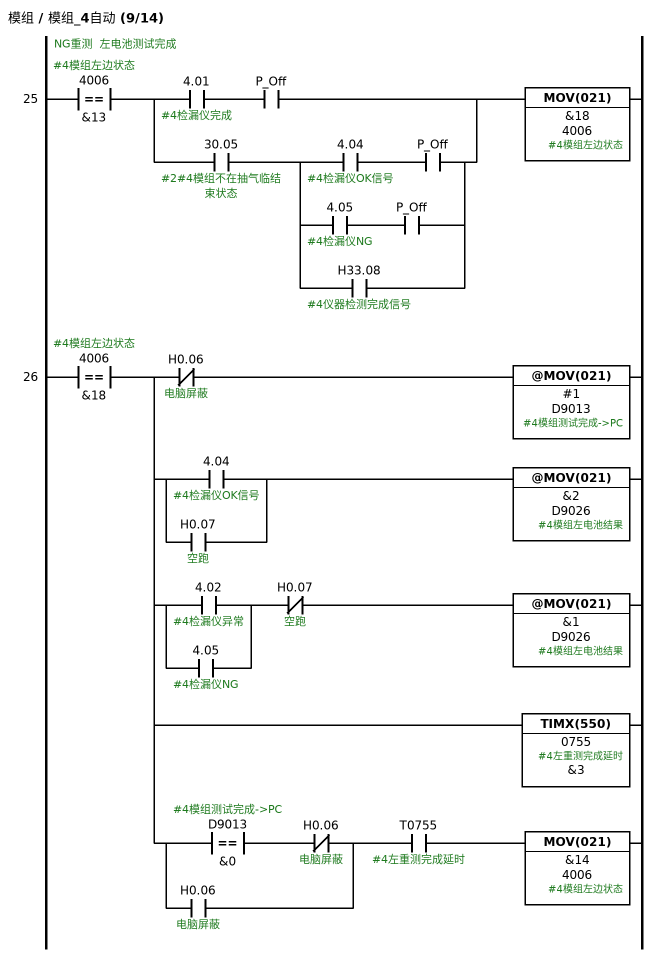
; [picture p257: 模组 / 模组_4自动, rungs 25-26]
; rung 25: NG重测  左电池测试完成
LD=(300) 4006 &13  ; #4模组左边状态
LD 4.01  ; #4检漏仪完成
AND P_Off
LD 30.05  ; #2#4模组不在抽气临结束状态  // 2018/5/29hy修改,所有模组不在临抽气结束状态下，测试模组测试完成后，给出停止测试信号
LD 4.04  ; #4检漏仪OK信号
AND P_Off
LD 4.05  ; #4检漏仪NG
AND P_Off
ORLD
OR H33.08  ; #4仪器检测完成信号
ANDLD
ORLD
ANDLD
MOV(021) &18 4006  ; #4模组左边状态
; rung 26
LD=(300) 4006 &18  ; #4模组左边状态
OUT TR0
ANDNOT H0.06  ; 电脑屏蔽
@MOV(021) #1 D9013  ; #4模组测试完成->PC
LD TR0
LD 4.04  ; #4检漏仪OK信号
OR H0.07  ; 空跑
ANDLD
@MOV(021) &2 D9026  ; #4模组左电池结果
LD TR0
LD 4.02  ; #4检漏仪异常
OR 4.05  ; #4检漏仪NG
ANDLD
ANDNOT H0.07  ; 空跑
@MOV(021) &1 D9026  ; #4模组左电池结果
LD TR0
TIMX(550) 0755 &3  ; #4左重测完成延时
LD=(300) D9013 &0  ; #4模组测试完成->PC
ANDNOT H0.06  ; 电脑屏蔽
OR H0.06  ; 电脑屏蔽
ANDLD
AND T0755  ; #4左重测完成延时
MOV(021) &14 4006  ; #4模组左边状态

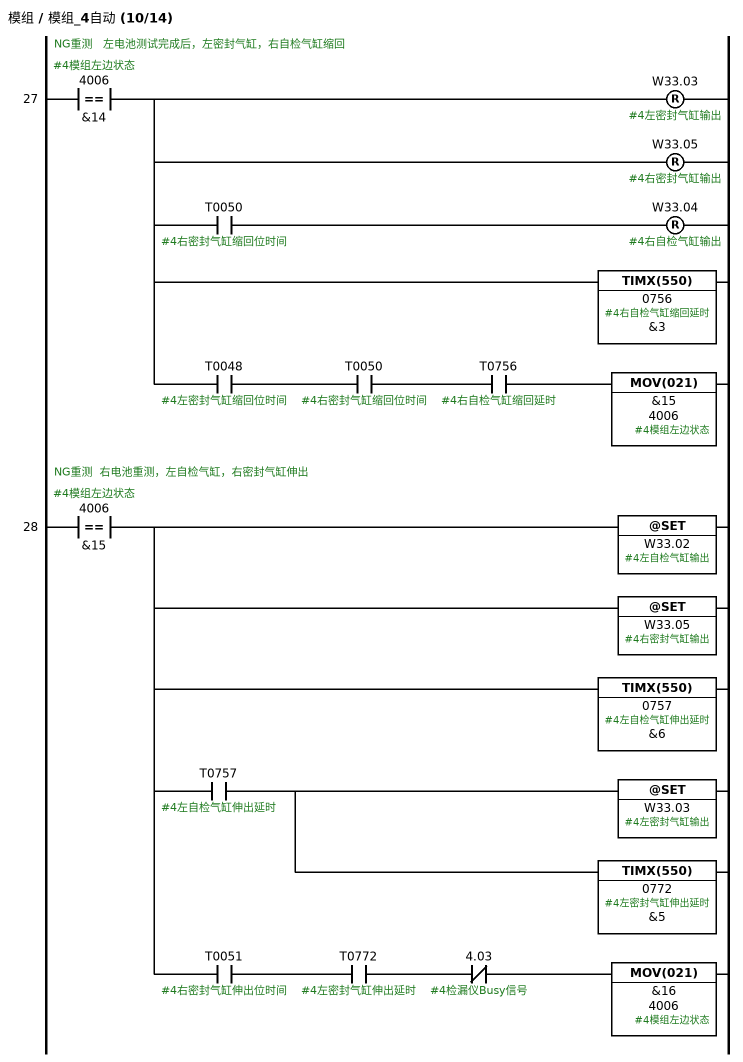
; rung 27: NG重测   左电池测试完成后，左密封气缸，右自检气缸缩回
LD=(300) 4006 &14  ; #4模组左边状态
OUT TR0
RSET W33.03  ; #4左密封气缸输出
RSET W33.05  ; #4右密封气缸输出
AND T0050  ; #4右密封气缸缩回位时间
RSET W33.04  ; #4右自检气缸输出
LD TR0
TIMX(550) 0756 &3  ; #4右自检气缸缩回延时
AND T0048  ; #4左密封气缸缩回位时间
AND T0050  ; #4右密封气缸缩回位时间
AND T0756  ; #4右自检气缸缩回延时
MOV(021) &15 4006  ; #4模组左边状态
; rung 28: NG重测  右电池重测，左自检气缸，右密封气缸伸出
LD=(300) 4006 &15  ; #4模组左边状态
OUT TR0
@SET W33.02  ; #4左自检气缸输出
@SET W33.05  ; #4右密封气缸输出
TIMX(550) 0757 &6  ; #4左自检气缸伸出延时
AND T0757  ; #4左自检气缸伸出延时
@SET W33.03  ; #4左密封气缸输出
TIMX(550) 0772 &5  ; #4左密封气缸伸出延时
LD TR0
AND T0051  ; #4右密封气缸伸出位时间
AND T0772  ; #4左密封气缸伸出延时
ANDNOT 4.03  ; #4检漏仪Busy信号
MOV(021) &16 4006  ; #4模组左边状态

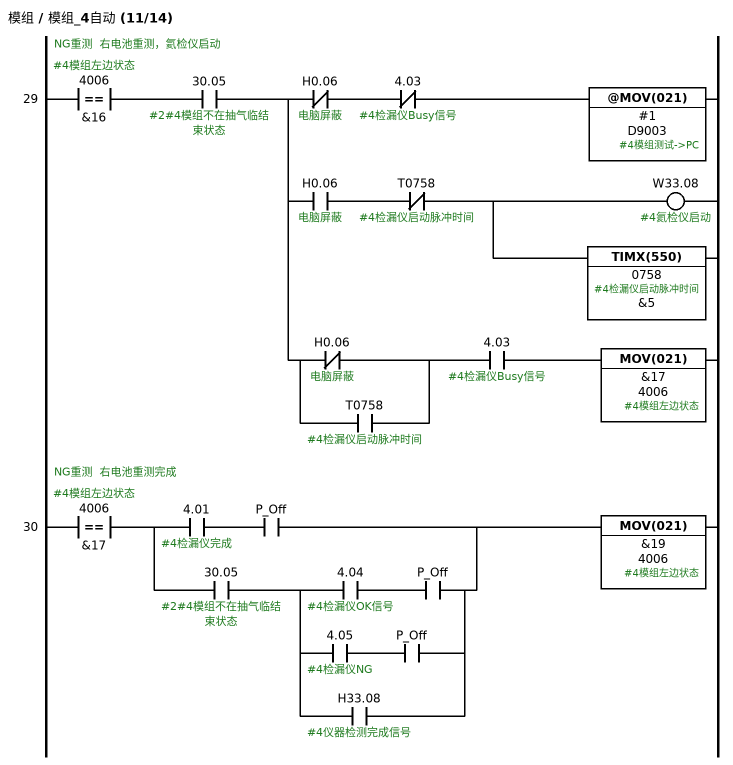
; rung 29: NG重测  右电池重测，氦检仪启动
LD=(300) 4006 &16  ; #4模组左边状态
AND 30.05  ; #2#4模组不在抽气临结束状态  // 2018/5/28hy修改 所有模组不在抽气临结束状态下，下一模组才能启动(防抽气NG)
OUT TR0
ANDNOT H0.06  ; 电脑屏蔽
ANDNOT 4.03  ; #4检漏仪Busy信号
@MOV(021) #1 D9003  ; #4模组测试->PC
LD TR0
AND H0.06  ; 电脑屏蔽
ANDNOT T0758  ; #4检漏仪启动脉冲时间
OUT W33.08  ; #4氦检仪启动
TIMX(550) 0758 &5  ; #4检漏仪启动脉冲时间
LD TR0
LDNOT H0.06  ; 电脑屏蔽
OR T0758  ; #4检漏仪启动脉冲时间
ANDLD
AND 4.03  ; #4检漏仪Busy信号
MOV(021) &17 4006  ; #4模组左边状态
; rung 30: NG重测  右电池重测完成
LD=(300) 4006 &17  ; #4模组左边状态
LD 4.01  ; #4检漏仪完成
AND P_Off
LD 30.05  ; #2#4模组不在抽气临结束状态
LD 4.04  ; #4检漏仪OK信号
AND P_Off
LD 4.05  ; #4检漏仪NG
AND P_Off
ORLD
OR H33.08  ; #4仪器检测完成信号
ANDLD
ORLD
ANDLD
MOV(021) &19 4006  ; #4模组左边状态

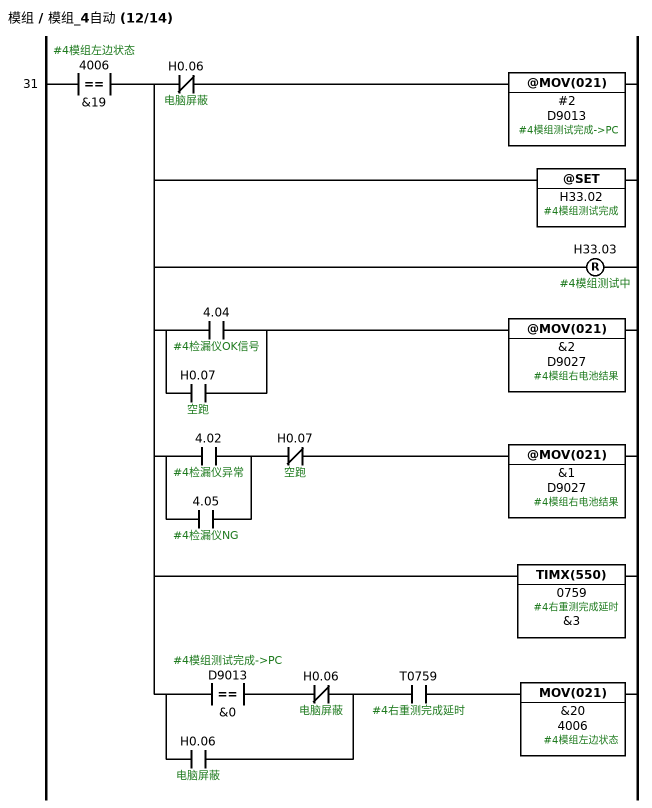
; rung 31
LD=(300) 4006 &19  ; #4模组左边状态
OUT TR0
ANDNOT H0.06  ; 电脑屏蔽
@MOV(021) #2 D9013  ; #4模组测试完成->PC
LD TR0
@SET H33.02  ; #4模组测试完成
RSET H33.03  ; #4模组测试中
LD 4.04  ; #4检漏仪OK信号
OR H0.07  ; 空跑
ANDLD
@MOV(021) &2 D9027  ; #4模组右电池结果
LD TR0
LD 4.02  ; #4检漏仪异常
OR 4.05  ; #4检漏仪NG
ANDLD
ANDNOT H0.07  ; 空跑
@MOV(021) &1 D9027  ; #4模组右电池结果
LD TR0
TIMX(550) 0759 &3  ; #4右重测完成延时
LD=(300) D9013 &0  ; #4模组测试完成->PC
ANDNOT H0.06  ; 电脑屏蔽
OR H0.06  ; 电脑屏蔽
ANDLD
AND T0759  ; #4右重测完成延时
MOV(021) &20 4006  ; #4模组左边状态

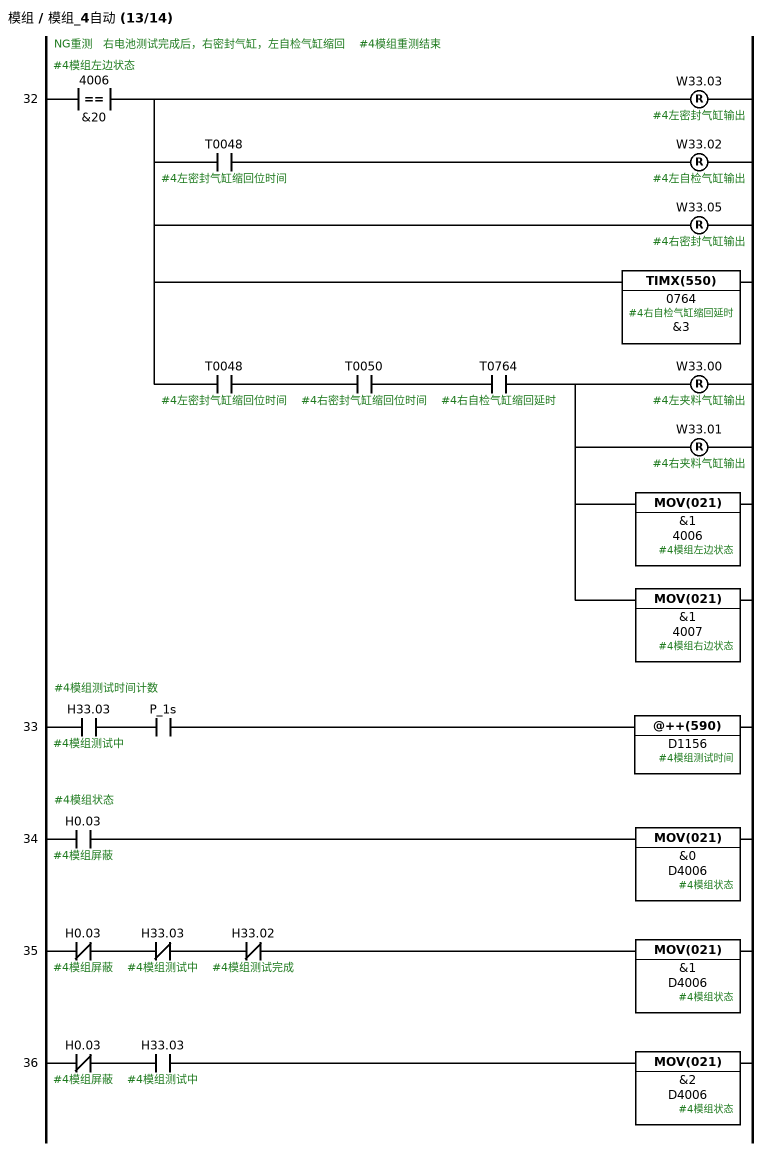
; rung 32: NG重测   右电池测试完成后，右密封气缸，左自检气缸缩回    #4模组重测结束
LD=(300) 4006 &20  ; #4模组左边状态
OUT TR0
RSET W33.03  ; #4左密封气缸输出
AND T0048  ; #4左密封气缸缩回位时间
RSET W33.02  ; #4左自检气缸输出
LD TR0
RSET W33.05  ; #4右密封气缸输出
TIMX(550) 0764 &3  ; #4右自检气缸缩回延时
AND T0048  ; #4左密封气缸缩回位时间
AND T0050  ; #4右密封气缸缩回位时间
AND T0764  ; #4右自检气缸缩回延时
RSET W33.00  ; #4左夹料气缸输出
RSET W33.01  ; #4右夹料气缸输出
MOV(021) &1 4006  ; #4模组左边状态
MOV(021) &1 4007  ; #4模组右边状态
; rung 33: #4模组测试时间计数
LD H33.03  ; #4模组测试中
AND P_1s
@++(590) D1156  ; #4模组测试时间
; rung 34: #4模组状态
LD H0.03  ; #4模组屏蔽
MOV(021) &0 D4006  ; #4模组状态
; rung 35
LDNOT H0.03  ; #4模组屏蔽
ANDNOT H33.03  ; #4模组测试中
ANDNOT H33.02  ; #4模组测试完成
MOV(021) &1 D4006  ; #4模组状态
; rung 36
LDNOT H0.03  ; #4模组屏蔽
AND H33.03  ; #4模组测试中
MOV(021) &2 D4006  ; #4模组状态

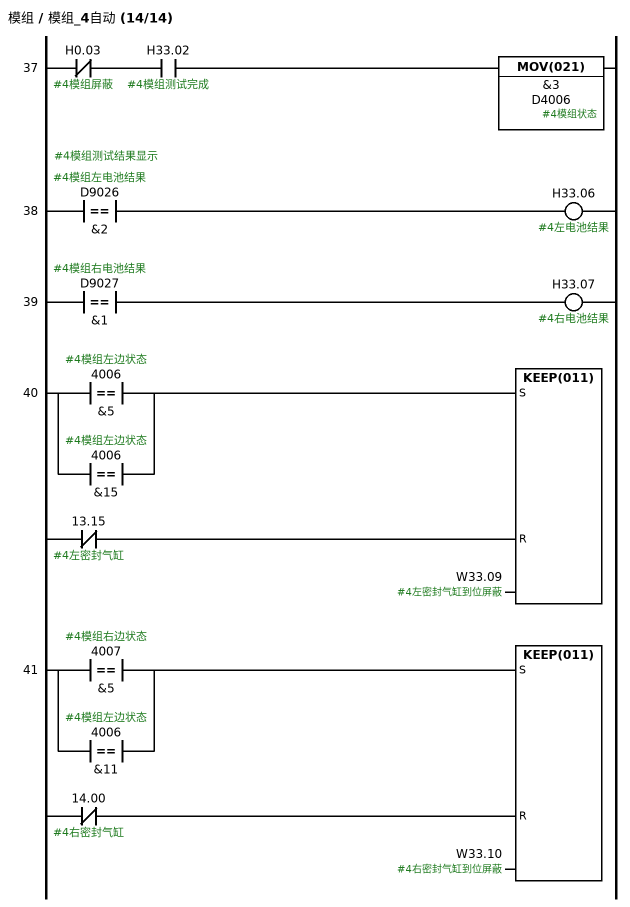
; rung 37
LDNOT H0.03  ; #4模组屏蔽
AND H33.02  ; #4模组测试完成
MOV(021) &3 D4006  ; #4模组状态
; rung 38: #4模组测试结果显示
LD=(300) D9026 &2  ; #4模组左电池结果
OUT H33.06  ; #4左电池结果
; rung 39
LD=(300) D9027 &1  ; #4模组右电池结果
OUT H33.07  ; #4右电池结果
; rung 40
LD=(300) 4006 &5  ; #4模组左边状态
OR=(300) 4006 &15  ; #4模组左边状态
LDNOT 13.15  ; #4左密封气缸
KEEP(011) W33.09  ; #4左密封气缸到位屏蔽
; rung 41
LD=(300) 4007 &5  ; #4模组右边状态
OR=(300) 4006 &11  ; #4模组左边状态
LDNOT 14.00  ; #4右密封气缸
KEEP(011) W33.10  ; #4右密封气缸到位屏蔽

### Section 外部输出

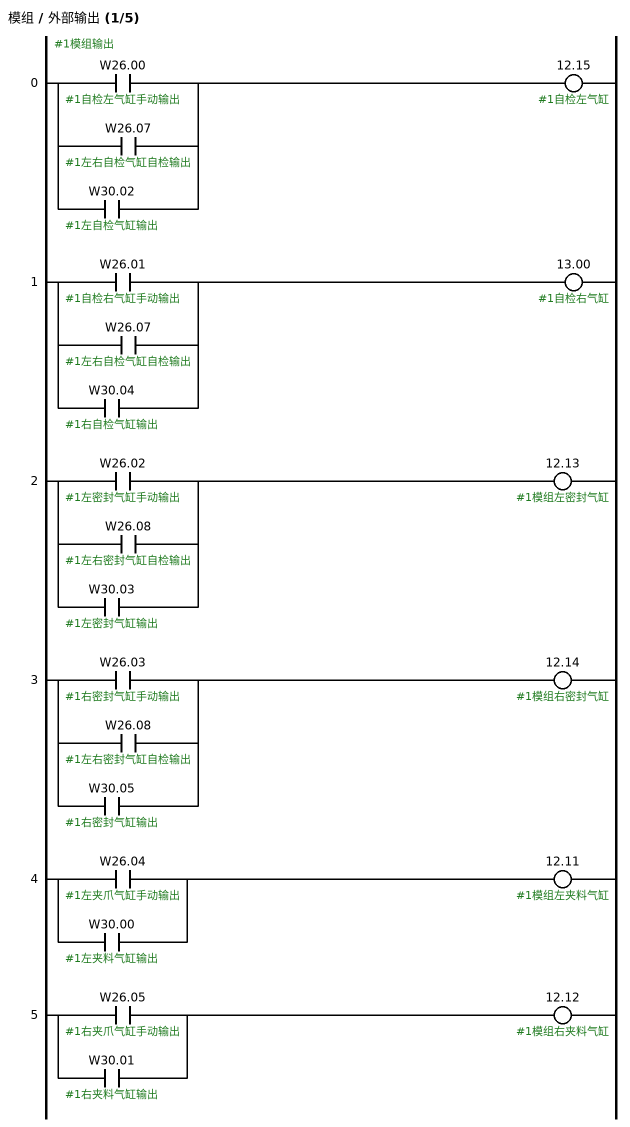
; rung 0: #1模组输出
LD W26.00  ; #1自检左气缸手动输出
OR W26.07  ; #1左右自检气缸自检输出
OR W30.02  ; #1左自检气缸输出
OUT 12.15  ; #1自检左气缸
; rung 1
LD W26.01  ; #1自检右气缸手动输出
OR W26.07  ; #1左右自检气缸自检输出
OR W30.04  ; #1右自检气缸输出
OUT 13.00  ; #1自检右气缸
; rung 2
LD W26.02  ; #1左密封气缸手动输出
OR W26.08  ; #1左右密封气缸自检输出
OR W30.03  ; #1左密封气缸输出
OUT 12.13  ; #1模组左密封气缸
; rung 3
LD W26.03  ; #1右密封气缸手动输出
OR W26.08  ; #1左右密封气缸自检输出
OR W30.05  ; #1右密封气缸输出
OUT 12.14  ; #1模组右密封气缸
; rung 4
LD W26.04  ; #1左夹爪气缸手动输出
OR W30.00  ; #1左夹料气缸输出
OUT 12.11  ; #1模组左夹料气缸
; rung 5
LD W26.05  ; #1右夹爪气缸手动输出
OR W30.01  ; #1右夹料气缸输出
OUT 12.12  ; #1模组右夹料气缸

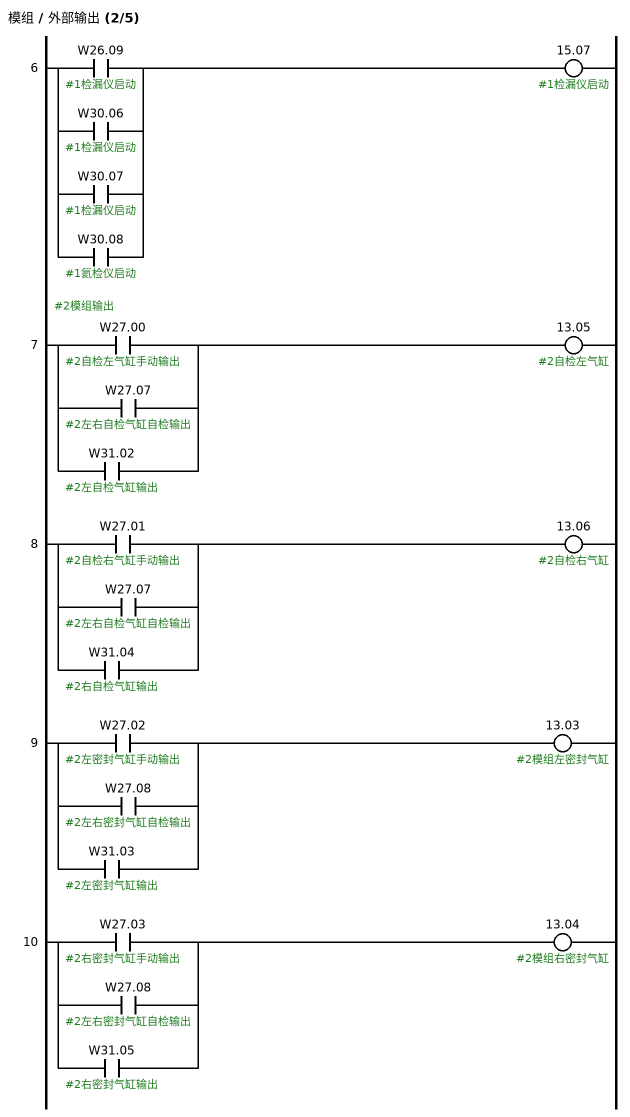
; rung 6
LD W26.09  ; #1检漏仪启动
OR W30.06  ; #1检漏仪启动
OR W30.07  ; #1检漏仪启动
OR W30.08  ; #1氦检仪启动
OUT 15.07  ; #1检漏仪启动
; rung 7: #2模组输出
LD W27.00  ; #2自检左气缸手动输出
OR W27.07  ; #2左右自检气缸自检输出
OR W31.02  ; #2左自检气缸输出
OUT 13.05  ; #2自检左气缸
; rung 8
LD W27.01  ; #2自检右气缸手动输出
OR W27.07  ; #2左右自检气缸自检输出
OR W31.04  ; #2右自检气缸输出
OUT 13.06  ; #2自检右气缸
; rung 9
LD W27.02  ; #2左密封气缸手动输出
OR W27.08  ; #2左右密封气缸自检输出
OR W31.03  ; #2左密封气缸输出
OUT 13.03  ; #2模组左密封气缸
; rung 10
LD W27.03  ; #2右密封气缸手动输出
OR W27.08  ; #2左右密封气缸自检输出
OR W31.05  ; #2右密封气缸输出
OUT 13.04  ; #2模组右密封气缸

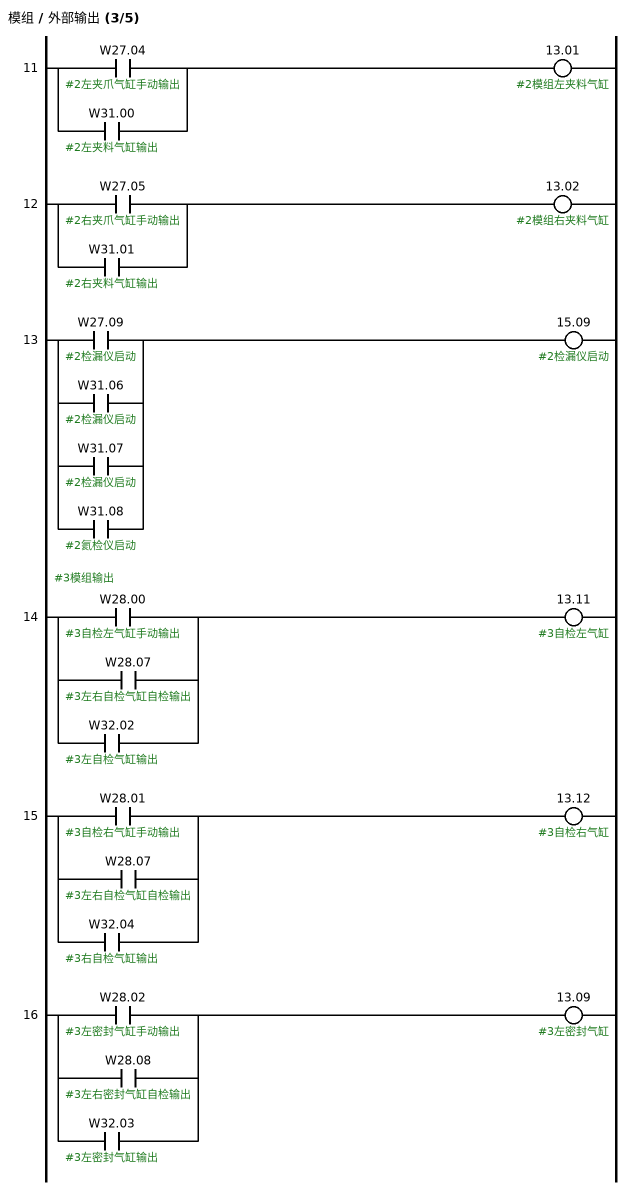
; rung 11
LD W27.04  ; #2左夹爪气缸手动输出
OR W31.00  ; #2左夹料气缸输出
OUT 13.01  ; #2模组左夹料气缸
; rung 12
LD W27.05  ; #2右夹爪气缸手动输出
OR W31.01  ; #2右夹料气缸输出
OUT 13.02  ; #2模组右夹料气缸
; rung 13
LD W27.09  ; #2检漏仪启动
OR W31.06  ; #2检漏仪启动
OR W31.07  ; #2检漏仪启动
OR W31.08  ; #2氦检仪启动
OUT 15.09  ; #2检漏仪启动
; rung 14: #3模组输出
LD W28.00  ; #3自检左气缸手动输出
OR W28.07  ; #3左右自检气缸自检输出
OR W32.02  ; #3左自检气缸输出
OUT 13.11  ; #3自检左气缸
; rung 15
LD W28.01  ; #3自检右气缸手动输出
OR W28.07  ; #3左右自检气缸自检输出
OR W32.04  ; #3右自检气缸输出
OUT 13.12  ; #3自检右气缸
; rung 16
LD W28.02  ; #3左密封气缸手动输出
OR W28.08  ; #3左右密封气缸自检输出
OR W32.03  ; #3左密封气缸输出
OUT 13.09  ; #3左密封气缸

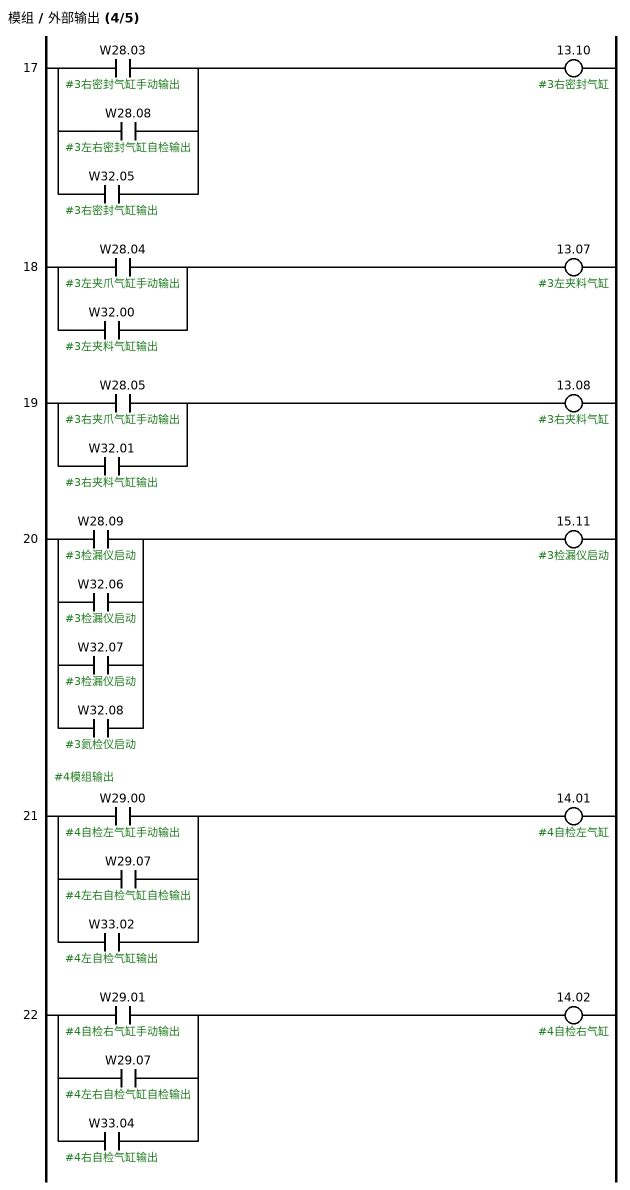
; rung 17
LD W28.03  ; #3右密封气缸手动输出
OR W28.08  ; #3左右密封气缸自检输出
OR W32.05  ; #3右密封气缸输出
OUT 13.10  ; #3右密封气缸
; rung 18
LD W28.04  ; #3左夹爪气缸手动输出
OR W32.00  ; #3左夹料气缸输出
OUT 13.07  ; #3左夹料气缸
; rung 19
LD W28.05  ; #3右夹爪气缸手动输出
OR W32.01  ; #3右夹料气缸输出
OUT 13.08  ; #3右夹料气缸
; rung 20
LD W28.09  ; #3检漏仪启动
OR W32.06  ; #3检漏仪启动
OR W32.07  ; #3检漏仪启动
OR W32.08  ; #3氦检仪启动
OUT 15.11  ; #3检漏仪启动
; rung 21: #4模组输出
LD W29.00  ; #4自检左气缸手动输出
OR W29.07  ; #4左右自检气缸自检输出
OR W33.02  ; #4左自检气缸输出
OUT 14.01  ; #4自检左气缸
; rung 22
LD W29.01  ; #4自检右气缸手动输出
OR W29.07  ; #4左右自检气缸自检输出
OR W33.04  ; #4右自检气缸输出
OUT 14.02  ; #4自检右气缸

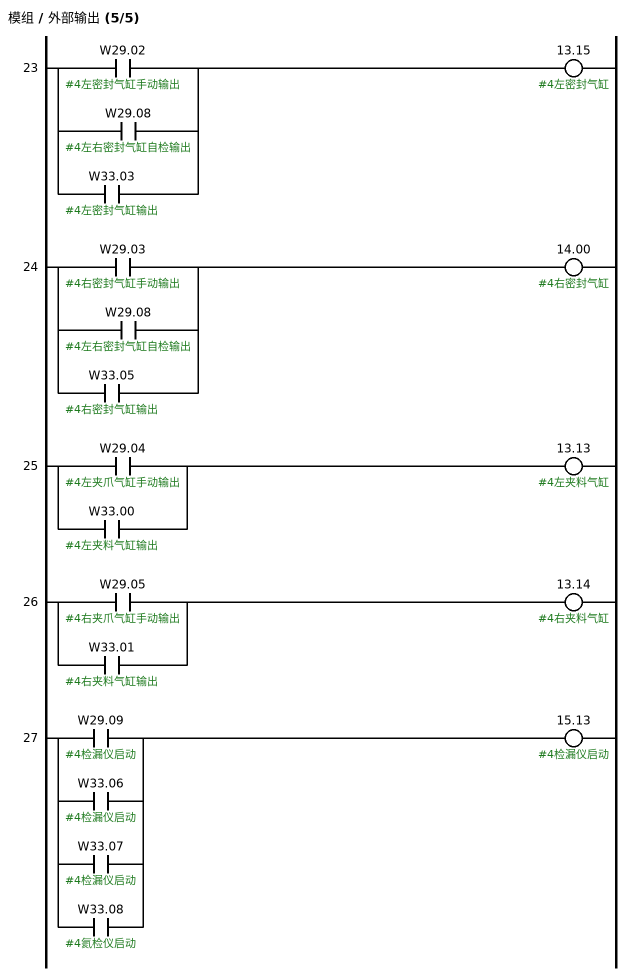
; rung 23
LD W29.02  ; #4左密封气缸手动输出
OR W29.08  ; #4左右密封气缸自检输出
OR W33.03  ; #4左密封气缸输出
OUT 13.15  ; #4左密封气缸
; rung 24
LD W29.03  ; #4右密封气缸手动输出
OR W29.08  ; #4左右密封气缸自检输出
OR W33.05  ; #4右密封气缸输出
OUT 14.00  ; #4右密封气缸
; rung 25
LD W29.04  ; #4左夹爪气缸手动输出
OR W33.00  ; #4左夹料气缸输出
OUT 13.13  ; #4左夹料气缸
; rung 26
LD W29.05  ; #4右夹爪气缸手动输出
OR W33.01  ; #4右夹料气缸输出
OUT 13.14  ; #4右夹料气缸
; rung 27
LD W29.09  ; #4检漏仪启动
OR W33.06  ; #4检漏仪启动
OR W33.07  ; #4检漏仪启动
OR W33.08  ; #4氦检仪启动
OUT 15.13  ; #4检漏仪启动

### Section 自动报警

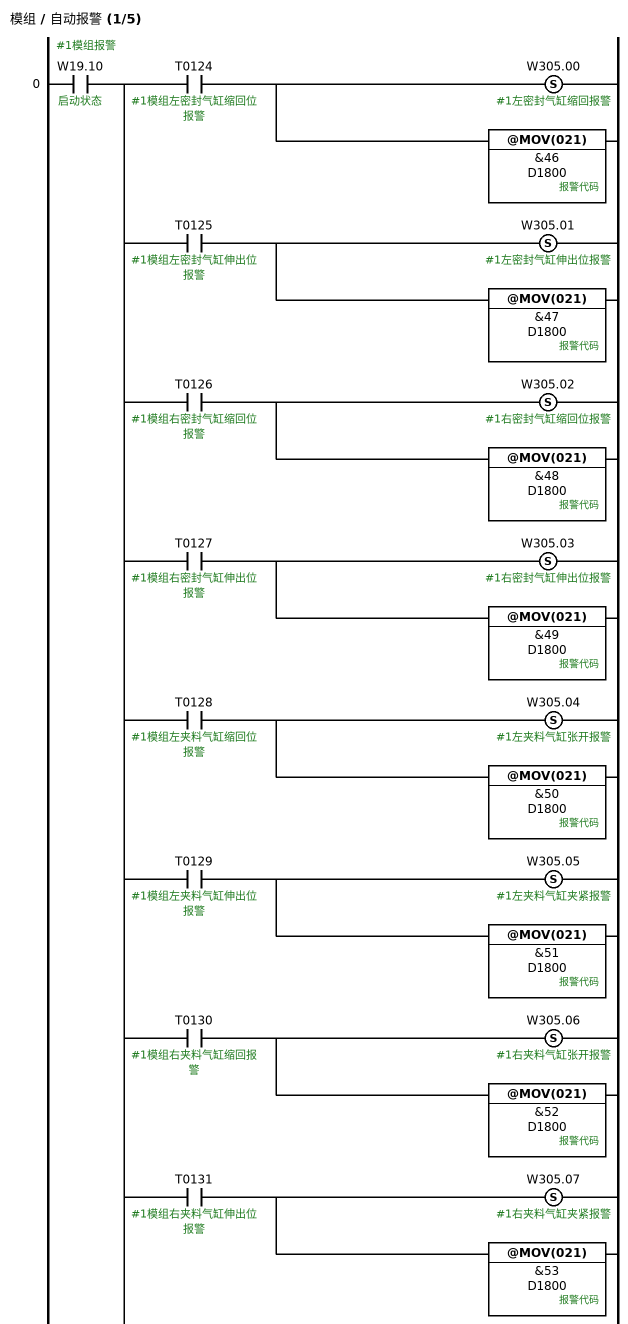

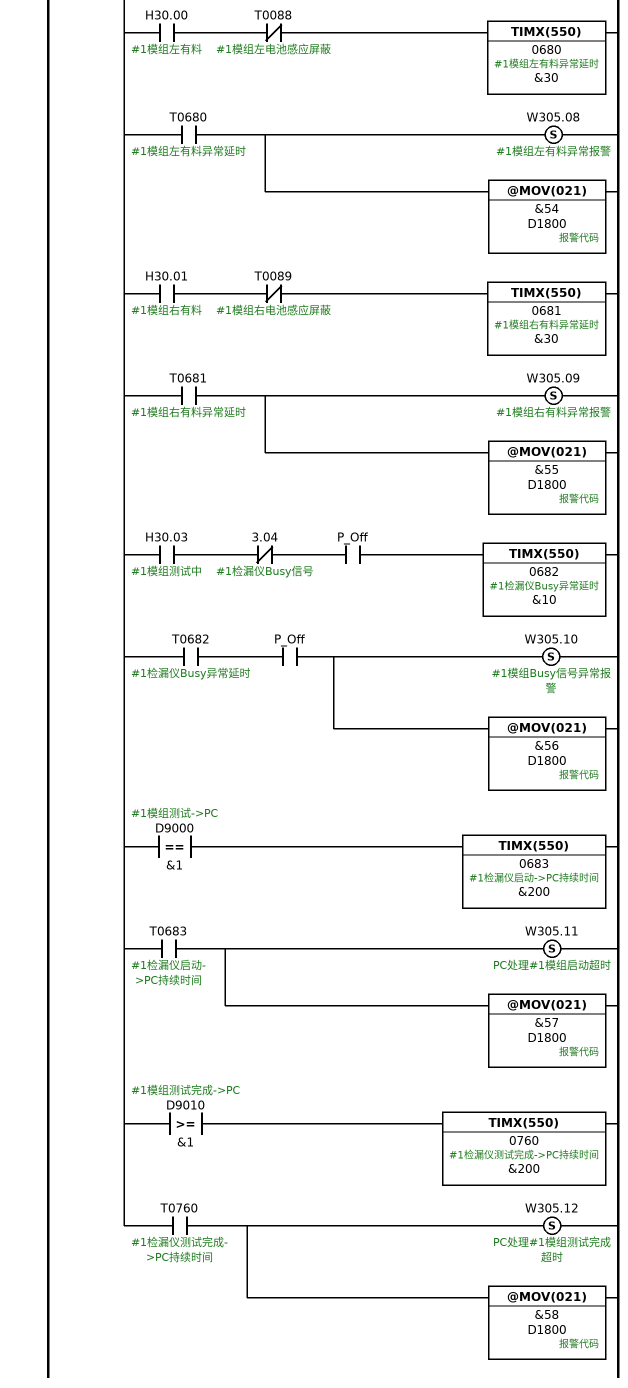
; rung 0: #1模组报警
LD W19.10  ; 启动状态
OUT TR0
AND T0124  ; #1模组左密封气缸缩回位报警
SET W305.00  ; #1左密封气缸缩回报警
@MOV(021) &46 D1800  ; 报警代码
LD TR0
AND T0125  ; #1模组左密封气缸伸出位报警
SET W305.01  ; #1左密封气缸伸出位报警
@MOV(021) &47 D1800  ; 报警代码
LD TR0
AND T0126  ; #1模组右密封气缸缩回位报警
SET W305.02  ; #1右密封气缸缩回位报警
@MOV(021) &48 D1800  ; 报警代码
LD TR0
AND T0127  ; #1模组右密封气缸伸出位报警
SET W305.03  ; #1右密封气缸伸出位报警
@MOV(021) &49 D1800  ; 报警代码
LD TR0
AND T0128  ; #1模组左夹料气缸缩回位报警
SET W305.04  ; #1左夹料气缸张开报警
@MOV(021) &50 D1800  ; 报警代码
LD TR0
AND T0129  ; #1模组左夹料气缸伸出位报警
SET W305.05  ; #1左夹料气缸夹紧报警
@MOV(021) &51 D1800  ; 报警代码
LD TR0
AND T0130  ; #1模组右夹料气缸缩回报警
SET W305.06  ; #1右夹料气缸张开报警
@MOV(021) &52 D1800  ; 报警代码
LD TR0
AND T0131  ; #1模组右夹料气缸伸出位报警
SET W305.07  ; #1右夹料气缸夹紧报警
@MOV(021) &53 D1800  ; 报警代码
LD TR0
AND H30.00  ; #1模组左有料
ANDNOT T0088  ; #1模组左电池感应屏蔽
TIMX(550) 0680 &30  ; #1模组左有料异常延时
LD TR0
AND T0680  ; #1模组左有料异常延时
SET W305.08  ; #1模组左有料异常报警
@MOV(021) &54 D1800  ; 报警代码
LD TR0
AND H30.01  ; #1模组右有料
ANDNOT T0089  ; #1模组右电池感应屏蔽
TIMX(550) 0681 &30  ; #1模组右有料异常延时
LD TR0
AND T0681  ; #1模组右有料异常延时
SET W305.09  ; #1模组右有料异常报警
@MOV(021) &55 D1800  ; 报警代码
LD TR0
AND H30.03  ; #1模组测试中
ANDNOT 3.04  ; #1检漏仪Busy信号
AND P_Off
TIMX(550) 0682 &10  ; #1检漏仪Busy异常延时
LD TR0
AND T0682  ; #1检漏仪Busy异常延时
AND P_Off
SET W305.10  ; #1模组Busy信号异常报警
@MOV(021) &56 D1800  ; 报警代码
LD TR0
AND=(300) D9000 &1  ; #1模组测试->PC
TIMX(550) 0683 &200  ; #1检漏仪启动->PC持续时间
LD TR0
AND T0683  ; #1检漏仪启动->PC持续时间
SET W305.11  ; PC处理#1模组启动超时
@MOV(021) &57 D1800  ; 报警代码
LD TR0
AND>=(325) D9010 &1  ; #1模组测试完成->PC
TIMX(550) 0760 &200  ; #1检漏仪测试完成->PC持续时间
LD TR0
AND T0760  ; #1检漏仪测试完成->PC持续时间
SET W305.12  ; PC处理#1模组测试完成超时
@MOV(021) &58 D1800  ; 报警代码

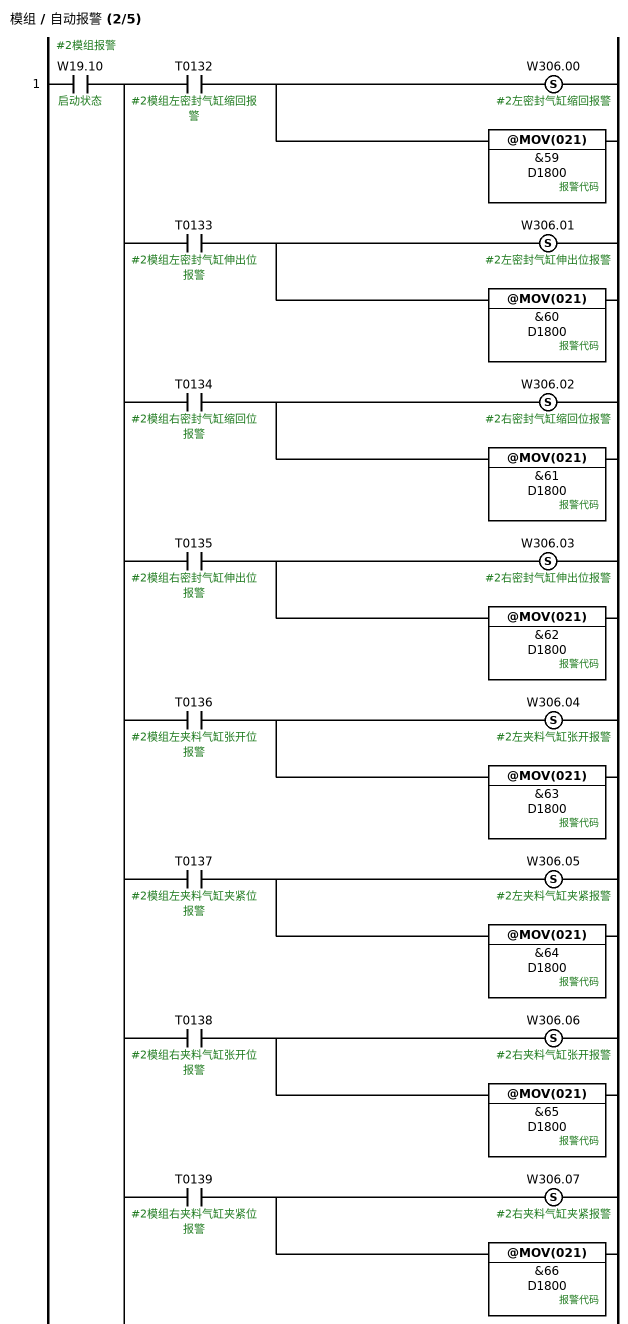

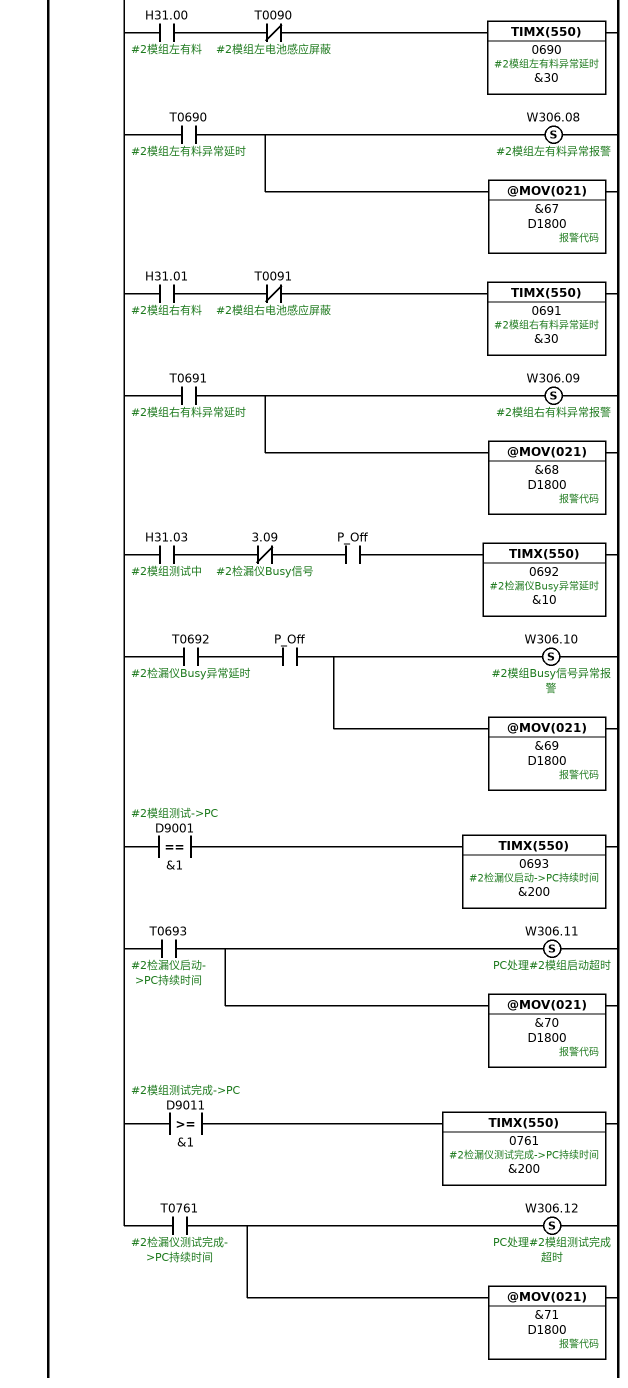
; rung 1: #2模组报警
LD W19.10  ; 启动状态
OUT TR0
AND T0132  ; #2模组左密封气缸缩回报警
SET W306.00  ; #2左密封气缸缩回报警
@MOV(021) &59 D1800  ; 报警代码
LD TR0
AND T0133  ; #2模组左密封气缸伸出位报警
SET W306.01  ; #2左密封气缸伸出位报警
@MOV(021) &60 D1800  ; 报警代码
LD TR0
AND T0134  ; #2模组右密封气缸缩回位报警
SET W306.02  ; #2右密封气缸缩回位报警
@MOV(021) &61 D1800  ; 报警代码
LD TR0
AND T0135  ; #2模组右密封气缸伸出位报警
SET W306.03  ; #2右密封气缸伸出位报警
@MOV(021) &62 D1800  ; 报警代码
LD TR0
AND T0136  ; #2模组左夹料气缸张开位报警
SET W306.04  ; #2左夹料气缸张开报警
@MOV(021) &63 D1800  ; 报警代码
LD TR0
AND T0137  ; #2模组左夹料气缸夹紧位报警
SET W306.05  ; #2左夹料气缸夹紧报警
@MOV(021) &64 D1800  ; 报警代码
LD TR0
AND T0138  ; #2模组右夹料气缸张开位报警
SET W306.06  ; #2右夹料气缸张开报警
@MOV(021) &65 D1800  ; 报警代码
LD TR0
AND T0139  ; #2模组右夹料气缸夹紧位报警
SET W306.07  ; #2右夹料气缸夹紧报警
@MOV(021) &66 D1800  ; 报警代码
LD TR0
AND H31.00  ; #2模组左有料
ANDNOT T0090  ; #2模组左电池感应屏蔽
TIMX(550) 0690 &30  ; #2模组左有料异常延时
LD TR0
AND T0690  ; #2模组左有料异常延时
SET W306.08  ; #2模组左有料异常报警
@MOV(021) &67 D1800  ; 报警代码
LD TR0
AND H31.01  ; #2模组右有料
ANDNOT T0091  ; #2模组右电池感应屏蔽
TIMX(550) 0691 &30  ; #2模组右有料异常延时
LD TR0
AND T0691  ; #2模组右有料异常延时
SET W306.09  ; #2模组右有料异常报警
@MOV(021) &68 D1800  ; 报警代码
LD TR0
AND H31.03  ; #2模组测试中
ANDNOT 3.09  ; #2检漏仪Busy信号
AND P_Off
TIMX(550) 0692 &10  ; #2检漏仪Busy异常延时
LD TR0
AND T0692  ; #2检漏仪Busy异常延时
AND P_Off
SET W306.10  ; #2模组Busy信号异常报警
@MOV(021) &69 D1800  ; 报警代码
LD TR0
AND=(300) D9001 &1  ; #2模组测试->PC
TIMX(550) 0693 &200  ; #2检漏仪启动->PC持续时间
LD TR0
AND T0693  ; #2检漏仪启动->PC持续时间
SET W306.11  ; PC处理#2模组启动超时
@MOV(021) &70 D1800  ; 报警代码
LD TR0
AND>=(325) D9011 &1  ; #2模组测试完成->PC
TIMX(550) 0761 &200  ; #2检漏仪测试完成->PC持续时间
LD TR0
AND T0761  ; #2检漏仪测试完成->PC持续时间
SET W306.12  ; PC处理#2模组测试完成超时
@MOV(021) &71 D1800  ; 报警代码

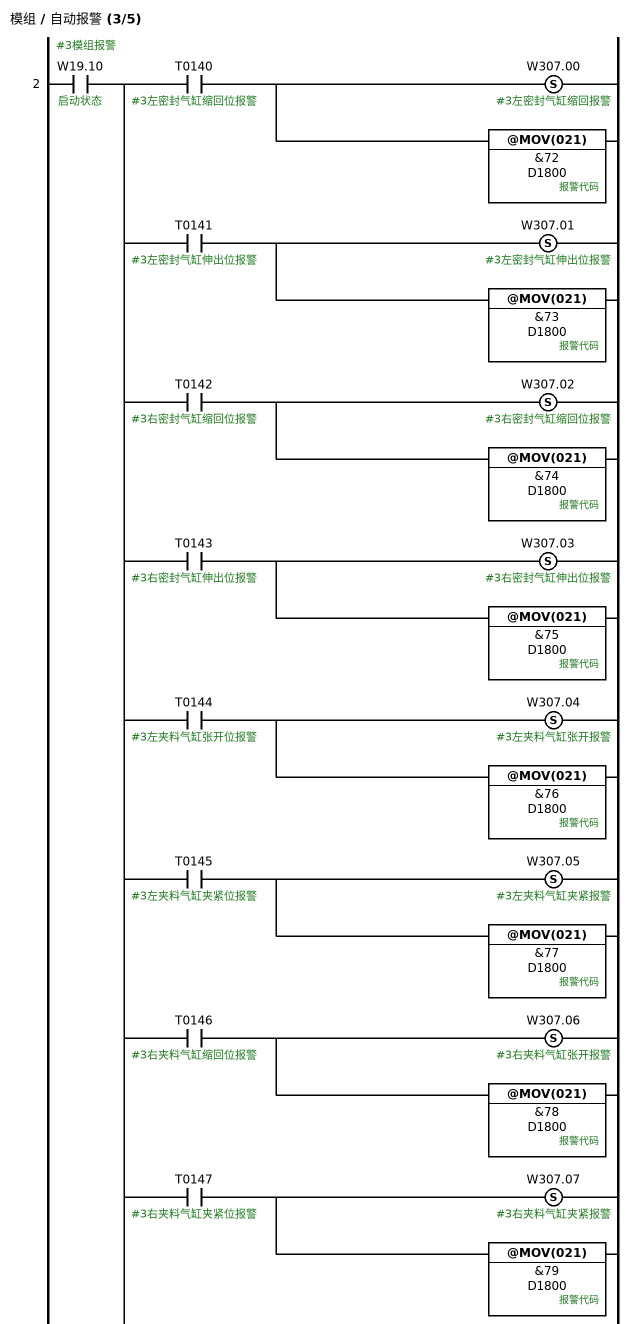

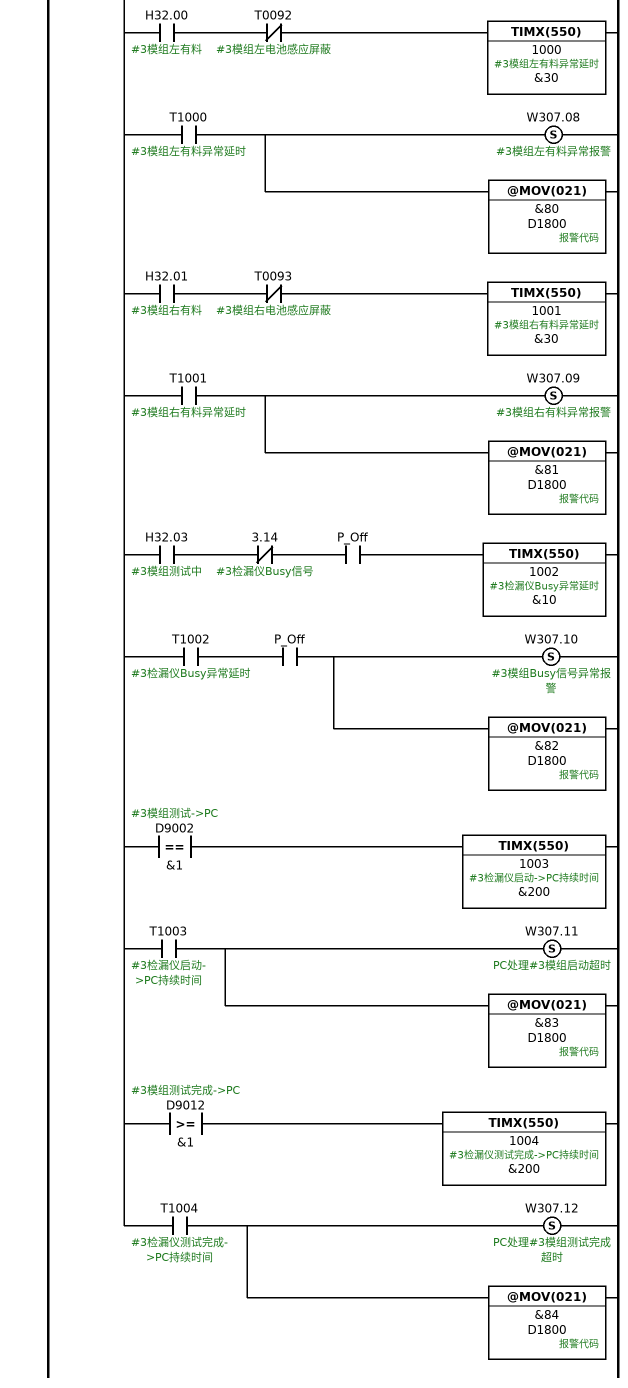
; rung 2: #3模组报警
LD W19.10  ; 启动状态
OUT TR0
AND T0140  ; #3左密封气缸缩回位报警
SET W307.00  ; #3左密封气缸缩回报警
@MOV(021) &72 D1800  ; 报警代码
LD TR0
AND T0141  ; #3左密封气缸伸出位报警
SET W307.01  ; #3左密封气缸伸出位报警
@MOV(021) &73 D1800  ; 报警代码
LD TR0
AND T0142  ; #3右密封气缸缩回位报警
SET W307.02  ; #3右密封气缸缩回位报警
@MOV(021) &74 D1800  ; 报警代码
LD TR0
AND T0143  ; #3右密封气缸伸出位报警
SET W307.03  ; #3右密封气缸伸出位报警
@MOV(021) &75 D1800  ; 报警代码
LD TR0
AND T0144  ; #3左夹料气缸张开位报警
SET W307.04  ; #3左夹料气缸张开报警
@MOV(021) &76 D1800  ; 报警代码
LD TR0
AND T0145  ; #3左夹料气缸夹紧位报警
SET W307.05  ; #3左夹料气缸夹紧报警
@MOV(021) &77 D1800  ; 报警代码
LD TR0
AND T0146  ; #3右夹料气缸缩回位报警
SET W307.06  ; #3右夹料气缸张开报警
@MOV(021) &78 D1800  ; 报警代码
LD TR0
AND T0147  ; #3右夹料气缸夹紧位报警
SET W307.07  ; #3右夹料气缸夹紧报警
@MOV(021) &79 D1800  ; 报警代码
LD TR0
AND H32.00  ; #3模组左有料
ANDNOT T0092  ; #3模组左电池感应屏蔽
TIMX(550) 1000 &30  ; #3模组左有料异常延时
LD TR0
AND T1000  ; #3模组左有料异常延时
SET W307.08  ; #3模组左有料异常报警
@MOV(021) &80 D1800  ; 报警代码
LD TR0
AND H32.01  ; #3模组右有料
ANDNOT T0093  ; #3模组右电池感应屏蔽
TIMX(550) 1001 &30  ; #3模组右有料异常延时
LD TR0
AND T1001  ; #3模组右有料异常延时
SET W307.09  ; #3模组右有料异常报警
@MOV(021) &81 D1800  ; 报警代码
LD TR0
AND H32.03  ; #3模组测试中
ANDNOT 3.14  ; #3检漏仪Busy信号
AND P_Off
TIMX(550) 1002 &10  ; #3检漏仪Busy异常延时
LD TR0
AND T1002  ; #3检漏仪Busy异常延时
AND P_Off
SET W307.10  ; #3模组Busy信号异常报警
@MOV(021) &82 D1800  ; 报警代码
LD TR0
AND=(300) D9002 &1  ; #3模组测试->PC
TIMX(550) 1003 &200  ; #3检漏仪启动->PC持续时间
LD TR0
AND T1003  ; #3检漏仪启动->PC持续时间
SET W307.11  ; PC处理#3模组启动超时
@MOV(021) &83 D1800  ; 报警代码
LD TR0
AND>=(325) D9012 &1  ; #3模组测试完成->PC
TIMX(550) 1004 &200  ; #3检漏仪测试完成->PC持续时间
LD TR0
AND T1004  ; #3检漏仪测试完成->PC持续时间
SET W307.12  ; PC处理#3模组测试完成超时
@MOV(021) &84 D1800  ; 报警代码

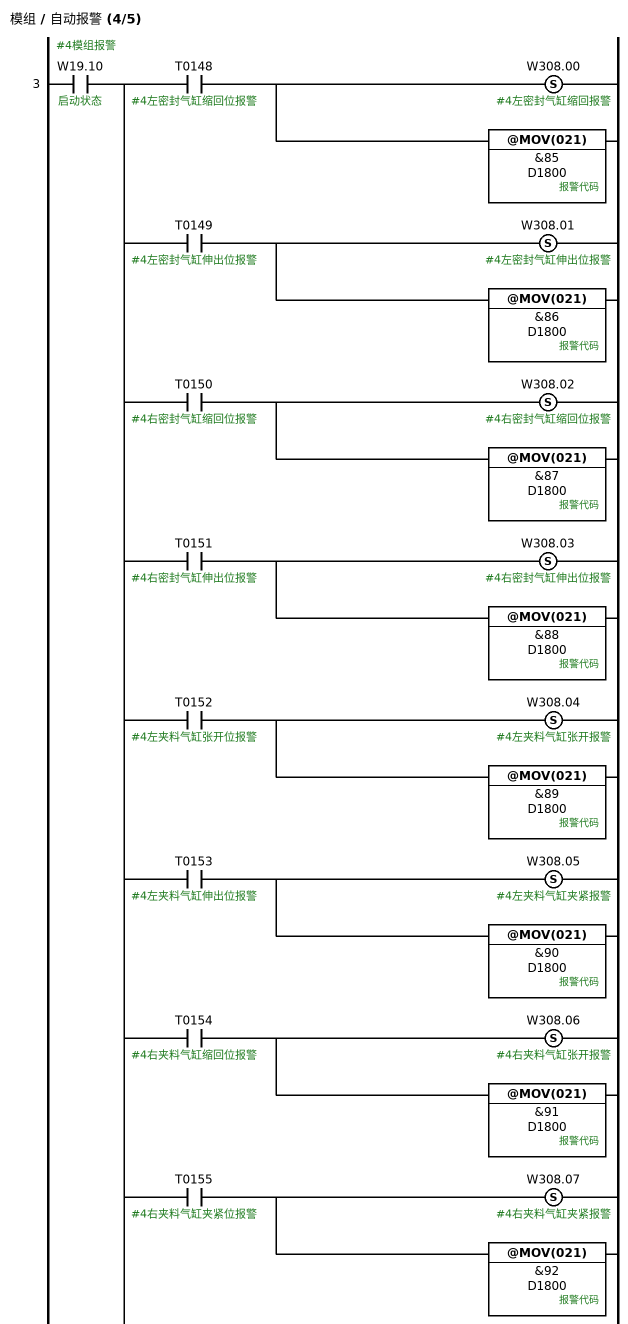

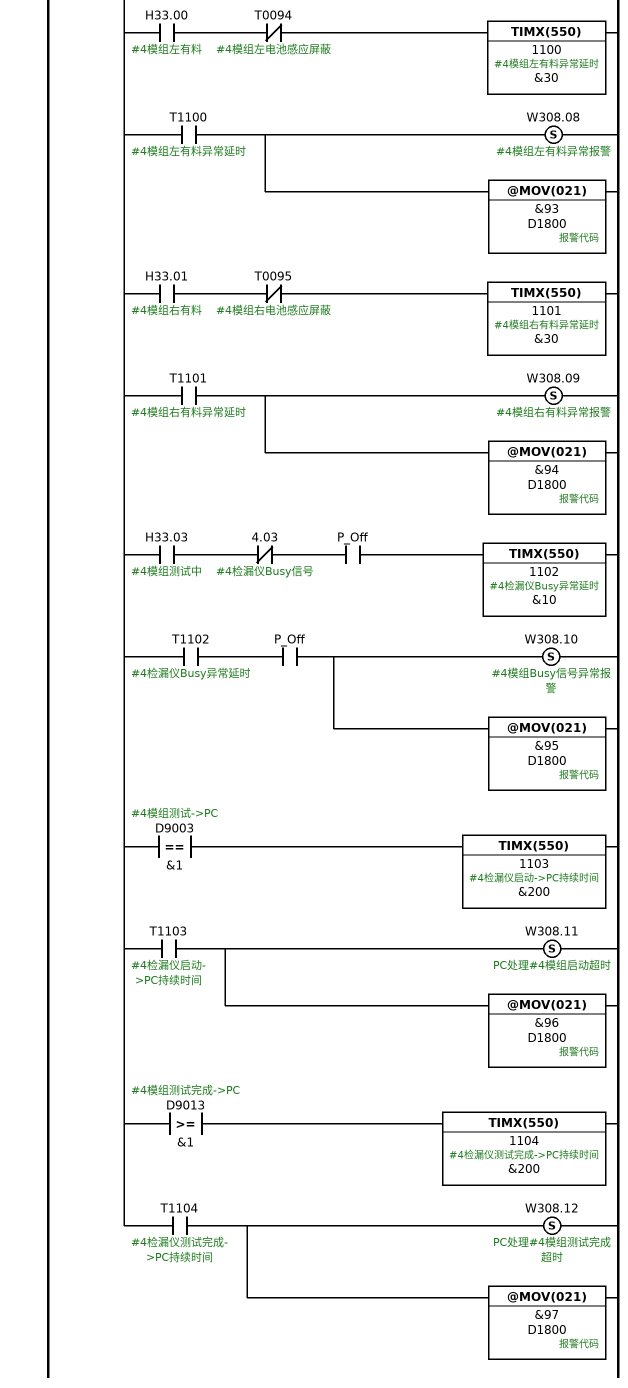
; rung 3: #4模组报警
LD W19.10  ; 启动状态
OUT TR0
AND T0148  ; #4左密封气缸缩回位报警
SET W308.00  ; #4左密封气缸缩回报警
@MOV(021) &85 D1800  ; 报警代码
LD TR0
AND T0149  ; #4左密封气缸伸出位报警
SET W308.01  ; #4左密封气缸伸出位报警
@MOV(021) &86 D1800  ; 报警代码
LD TR0
AND T0150  ; #4右密封气缸缩回位报警
SET W308.02  ; #4右密封气缸缩回位报警
@MOV(021) &87 D1800  ; 报警代码
LD TR0
AND T0151  ; #4右密封气缸伸出位报警
SET W308.03  ; #4右密封气缸伸出位报警
@MOV(021) &88 D1800  ; 报警代码
LD TR0
AND T0152  ; #4左夹料气缸张开位报警
SET W308.04  ; #4左夹料气缸张开报警
@MOV(021) &89 D1800  ; 报警代码
LD TR0
AND T0153  ; #4左夹料气缸伸出位报警
SET W308.05  ; #4左夹料气缸夹紧报警
@MOV(021) &90 D1800  ; 报警代码
LD TR0
AND T0154  ; #4右夹料气缸缩回位报警
SET W308.06  ; #4右夹料气缸张开报警
@MOV(021) &91 D1800  ; 报警代码
LD TR0
AND T0155  ; #4右夹料气缸夹紧位报警
SET W308.07  ; #4右夹料气缸夹紧报警
@MOV(021) &92 D1800  ; 报警代码
LD TR0
AND H33.00  ; #4模组左有料
ANDNOT T0094  ; #4模组左电池感应屏蔽
TIMX(550) 1100 &30  ; #4模组左有料异常延时
LD TR0
AND T1100  ; #4模组左有料异常延时
SET W308.08  ; #4模组左有料异常报警
@MOV(021) &93 D1800  ; 报警代码
LD TR0
AND H33.01  ; #4模组右有料
ANDNOT T0095  ; #4模组右电池感应屏蔽
TIMX(550) 1101 &30  ; #4模组右有料异常延时
LD TR0
AND T1101  ; #4模组右有料异常延时
SET W308.09  ; #4模组右有料异常报警
@MOV(021) &94 D1800  ; 报警代码
LD TR0
AND H33.03  ; #4模组测试中
ANDNOT 4.03  ; #4检漏仪Busy信号
AND P_Off
TIMX(550) 1102 &10  ; #4检漏仪Busy异常延时
LD TR0
AND T1102  ; #4检漏仪Busy异常延时
AND P_Off
SET W308.10  ; #4模组Busy信号异常报警
@MOV(021) &95 D1800  ; 报警代码
LD TR0
AND=(300) D9003 &1  ; #4模组测试->PC
TIMX(550) 1103 &200  ; #4检漏仪启动->PC持续时间
LD TR0
AND T1103  ; #4检漏仪启动->PC持续时间
SET W308.11  ; PC处理#4模组启动超时
@MOV(021) &96 D1800  ; 报警代码
LD TR0
AND>=(325) D9013 &1  ; #4模组测试完成->PC
TIMX(550) 1104 &200  ; #4检漏仪测试完成->PC持续时间
LD TR0
AND T1104  ; #4检漏仪测试完成->PC持续时间
SET W308.12  ; PC处理#4模组测试完成超时
@MOV(021) &97 D1800  ; 报警代码

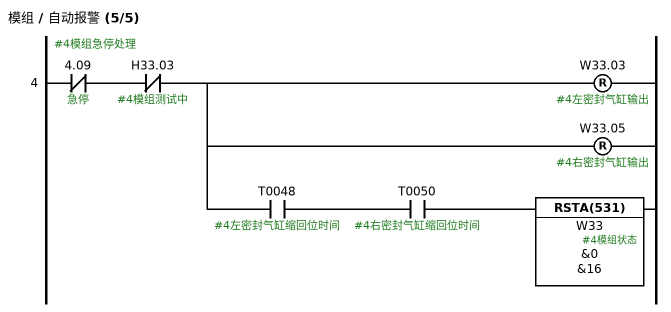
; rung 4: #4模组急停处理
LDNOT 4.09  ; 急停
ANDNOT H33.03  ; #4模组测试中
RSET W33.03  ; #4左密封气缸输出
RSET W33.05  ; #4右密封气缸输出
AND T0048  ; #4左密封气缸缩回位时间
AND T0050  ; #4右密封气缸缩回位时间
RSTA(531) W33 &0 &16  ; #4模组状态

### Section 模组复位

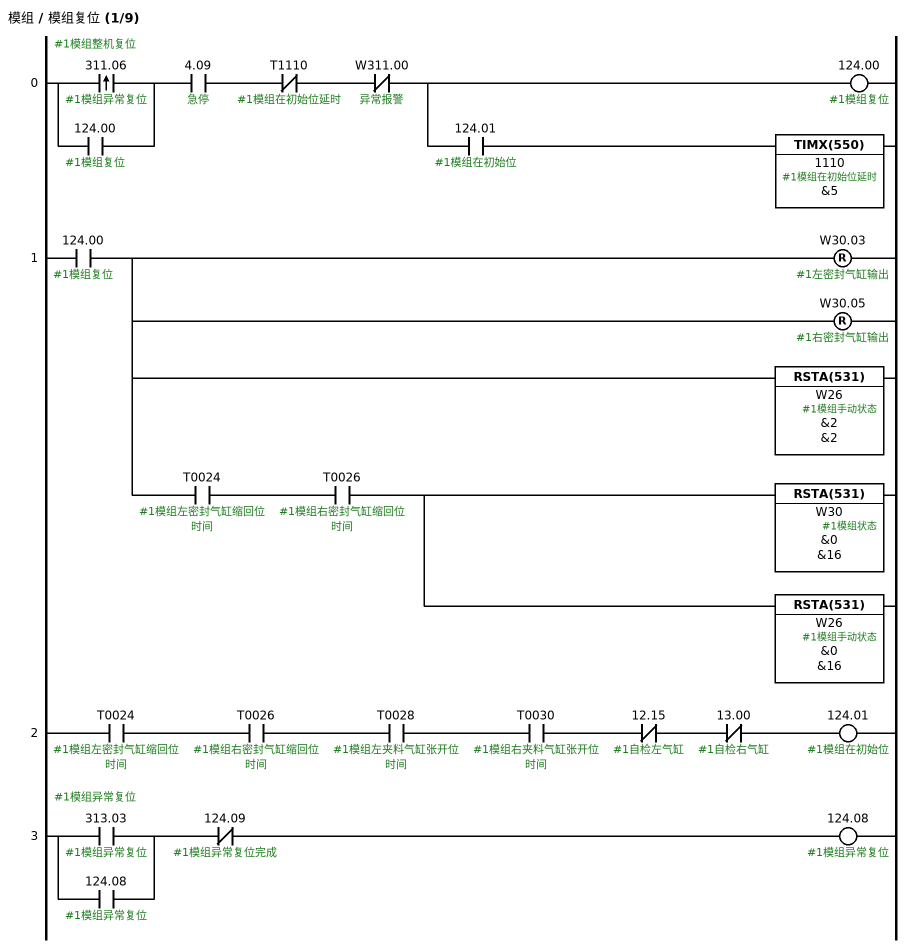
; rung 0: #1模组整机复位
@LD 311.06  ; #1模组异常复位
OR 124.00  ; #1模组复位
AND 4.09  ; 急停
ANDNOT T1110  ; #1模组在初始位延时
ANDNOT W311.00  ; 异常报警
OUT 124.00  ; #1模组复位
AND 124.01  ; #1模组在初始位
TIMX(550) 1110 &5  ; #1模组在初始位延时
; rung 1
LD 124.00  ; #1模组复位
RSET W30.03  ; #1左密封气缸输出
RSET W30.05  ; #1右密封气缸输出
RSTA(531) W26 &2 &2  ; #1模组手动状态
AND T0024  ; #1模组左密封气缸缩回位时间
AND T0026  ; #1模组右密封气缸缩回位时间
RSTA(531) W30 &0 &16  ; #1模组状态
RSTA(531) W26 &0 &16  ; #1模组手动状态
; rung 2
LD T0024  ; #1模组左密封气缸缩回位时间
AND T0026  ; #1模组右密封气缸缩回位时间
AND T0028  ; #1模组左夹料气缸张开位时间
AND T0030  ; #1模组右夹料气缸张开位时间
ANDNOT 12.15  ; #1自检左气缸
ANDNOT 13.00  ; #1自检右气缸
OUT 124.01  ; #1模组在初始位
; rung 3: #1模组异常复位
LD 313.03  ; #1模组异常复位
OR 124.08  ; #1模组异常复位
ANDNOT 124.09  ; #1模组异常复位完成
OUT 124.08  ; #1模组异常复位

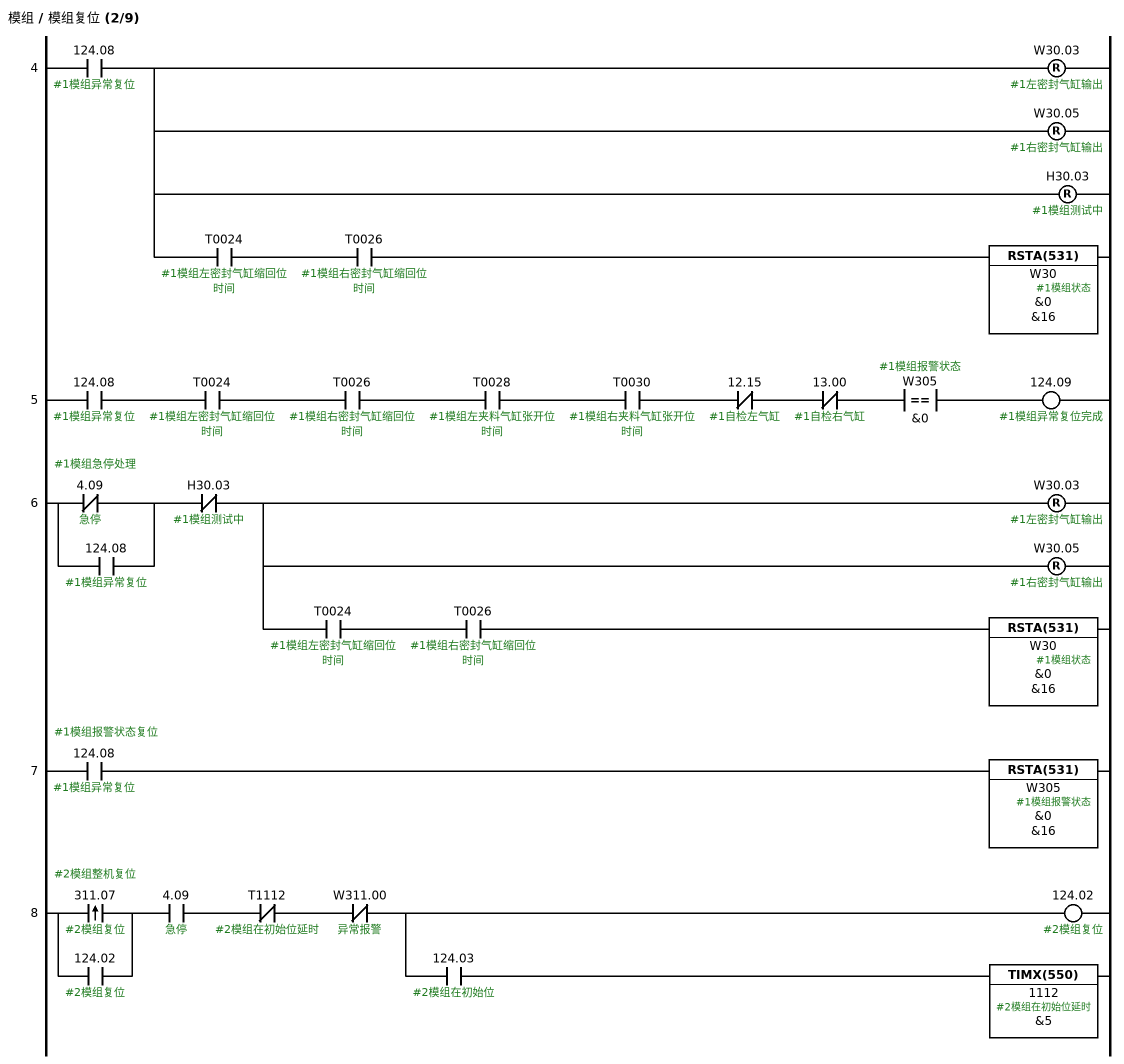
; rung 4
LD 124.08  ; #1模组异常复位
RSET W30.03  ; #1左密封气缸输出
RSET W30.05  ; #1右密封气缸输出
RSET H30.03  ; #1模组测试中
AND T0024  ; #1模组左密封气缸缩回位时间
AND T0026  ; #1模组右密封气缸缩回位时间
RSTA(531) W30 &0 &16  ; #1模组状态
; rung 5
LD 124.08  ; #1模组异常复位
AND T0024  ; #1模组左密封气缸缩回位时间
AND T0026  ; #1模组右密封气缸缩回位时间
AND T0028  ; #1模组左夹料气缸张开位时间
AND T0030  ; #1模组右夹料气缸张开位时间
ANDNOT 12.15  ; #1自检左气缸
ANDNOT 13.00  ; #1自检右气缸
AND=(300) W305 &0  ; #1模组报警状态
OUT 124.09  ; #1模组异常复位完成
; rung 6: #1模组急停处理
LDNOT 4.09  ; 急停
OR 124.08  ; #1模组异常复位
ANDNOT H30.03  ; #1模组测试中
RSET W30.03  ; #1左密封气缸输出
RSET W30.05  ; #1右密封气缸输出
AND T0024  ; #1模组左密封气缸缩回位时间
AND T0026  ; #1模组右密封气缸缩回位时间
RSTA(531) W30 &0 &16  ; #1模组状态
; rung 7: #1模组报警状态复位
LD 124.08  ; #1模组异常复位
RSTA(531) W305 &0 &16  ; #1模组报警状态
; rung 8: #2模组整机复位
@LD 311.07  ; #2模组复位
OR 124.02  ; #2模组复位
AND 4.09  ; 急停
ANDNOT T1112  ; #2模组在初始位延时
ANDNOT W311.00  ; 异常报警
OUT 124.02  ; #2模组复位
AND 124.03  ; #2模组在初始位
TIMX(550) 1112 &5  ; #2模组在初始位延时

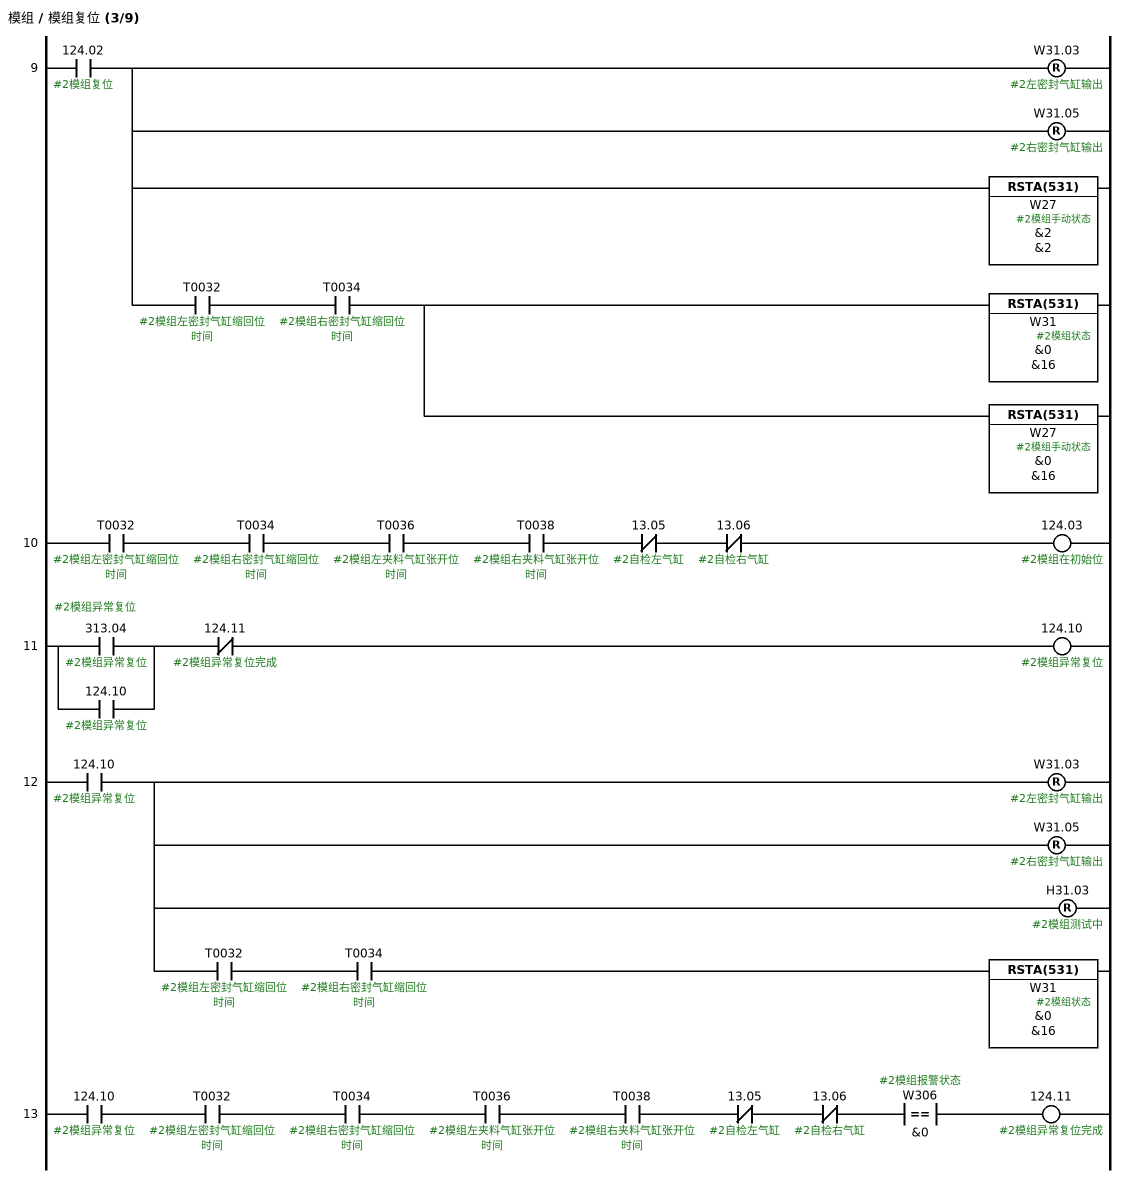
; rung 9
LD 124.02  ; #2模组复位
RSET W31.03  ; #2左密封气缸输出
RSET W31.05  ; #2右密封气缸输出
RSTA(531) W27 &2 &2  ; #2模组手动状态
AND T0032  ; #2模组左密封气缸缩回位时间
AND T0034  ; #2模组右密封气缸缩回位时间
RSTA(531) W31 &0 &16  ; #2模组状态
RSTA(531) W27 &0 &16  ; #2模组手动状态
; rung 10
LD T0032  ; #2模组左密封气缸缩回位时间
AND T0034  ; #2模组右密封气缸缩回位时间
AND T0036  ; #2模组左夹料气缸张开位时间
AND T0038  ; #2模组右夹料气缸张开位时间
ANDNOT 13.05  ; #2自检左气缸
ANDNOT 13.06  ; #2自检右气缸
OUT 124.03  ; #2模组在初始位
; rung 11: #2模组异常复位
LD 313.04  ; #2模组异常复位
OR 124.10  ; #2模组异常复位
ANDNOT 124.11  ; #2模组异常复位完成
OUT 124.10  ; #2模组异常复位
; rung 12
LD 124.10  ; #2模组异常复位
RSET W31.03  ; #2左密封气缸输出
RSET W31.05  ; #2右密封气缸输出
RSET H31.03  ; #2模组测试中
AND T0032  ; #2模组左密封气缸缩回位时间
AND T0034  ; #2模组右密封气缸缩回位时间
RSTA(531) W31 &0 &16  ; #2模组状态
; rung 13
LD 124.10  ; #2模组异常复位
AND T0032  ; #2模组左密封气缸缩回位时间
AND T0034  ; #2模组右密封气缸缩回位时间
AND T0036  ; #2模组左夹料气缸张开位时间
AND T0038  ; #2模组右夹料气缸张开位时间
ANDNOT 13.05  ; #2自检左气缸
ANDNOT 13.06  ; #2自检右气缸
AND=(300) W306 &0  ; #2模组报警状态
OUT 124.11  ; #2模组异常复位完成

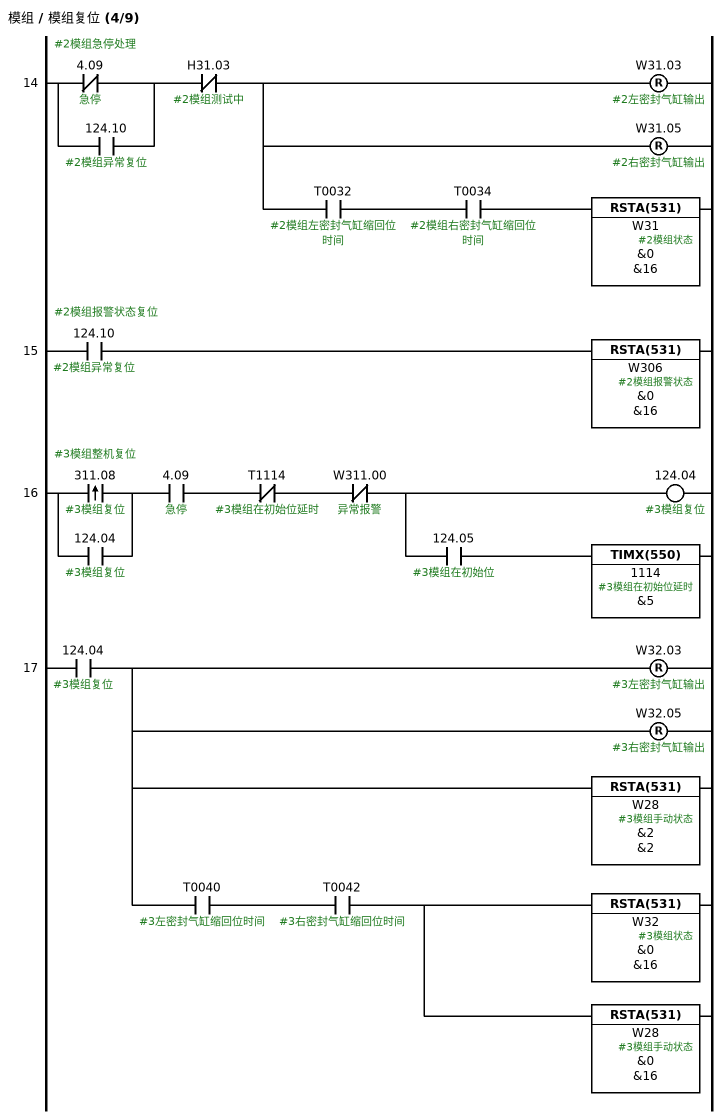
; rung 14: #2模组急停处理
LDNOT 4.09  ; 急停
OR 124.10  ; #2模组异常复位
ANDNOT H31.03  ; #2模组测试中
RSET W31.03  ; #2左密封气缸输出
RSET W31.05  ; #2右密封气缸输出
AND T0032  ; #2模组左密封气缸缩回位时间
AND T0034  ; #2模组右密封气缸缩回位时间
RSTA(531) W31 &0 &16  ; #2模组状态
; rung 15: #2模组报警状态复位
LD 124.10  ; #2模组异常复位
RSTA(531) W306 &0 &16  ; #2模组报警状态
; rung 16: #3模组整机复位
@LD 311.08  ; #3模组复位
OR 124.04  ; #3模组复位
AND 4.09  ; 急停
ANDNOT T1114  ; #3模组在初始位延时
ANDNOT W311.00  ; 异常报警
OUT 124.04  ; #3模组复位
AND 124.05  ; #3模组在初始位
TIMX(550) 1114 &5  ; #3模组在初始位延时
; rung 17
LD 124.04  ; #3模组复位
RSET W32.03  ; #3左密封气缸输出
RSET W32.05  ; #3右密封气缸输出
RSTA(531) W28 &2 &2  ; #3模组手动状态
AND T0040  ; #3左密封气缸缩回位时间
AND T0042  ; #3右密封气缸缩回位时间
RSTA(531) W32 &0 &16  ; #3模组状态
RSTA(531) W28 &0 &16  ; #3模组手动状态

